FUNCTION_BLOCK Stage4 (* Template for a Basic Function Block Type *)
  (* Standard: 61499-2 *)
  (* Version 1.0, 2021-06-20, HP *)
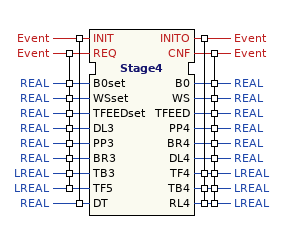
  EVENT_INPUT
    INIT WITH DT; (* Initialization Request *)
    REQ WITH B0set, WSset, TFEEDset, DL3, PP3, BR3, TB3, TF5; (* Normal Execution Request *)
  END_EVENT
  EVENT_OUTPUT
    INITO WITH TB4, TF4, RL4; (* Initialization Confirm *)
    CNF WITH TB4, DL4, TF4, BR4, PP4, RL4, B0, WS, TFEED; (* Execution Confirmation *)
  END_EVENT
  VAR_INPUT
    B0set : REAL;
    WSset : REAL;
    TFEEDset : REAL;
    DL3 : REAL;
    PP3 : REAL;
    BR3 : REAL;
    TB3 : LREAL;
    TF5 : LREAL;
    DT : REAL;
  END_VAR
  VAR_OUTPUT
    B0 : REAL;
    WS : REAL;
    TFEED : REAL;
    PP4 : REAL;
    BR4 : REAL;
    DL4 : REAL;
    TF4 : LREAL;
    TB4 : LREAL;
    RL4 : LREAL;
  END_VAR
  VAR
    AB : REAL; (* internal variabel *)
    UU : REAL;
    TREF : REAL;
    AD : REAL;
    AHC : REAL;
    AHR : REAL;
    AS : REAL;
    REC : REAL;
    WN : REAL;
    WN_1 : REAL;
    XKN : REAL;
    C1 : REAL;
    HS : REAL;
    G : REAL;
    W1 : REAL;
    TFREC : REAL;
    TS : REAL;
    DTS : REAL;
    TF4_last : REAL;
    RL4_last : REAL;
    TB4_last : REAL;
    USS : REAL;
    RHOB : REAL;
    CPB : REAL;
    CPF : REAL;
    FMW : REAL;
    HLV : REAL;
    HV : REAL;
    BPR : REAL;
    FMC : REAL;
    U : REAL;
    A : REAL;
    B : REAL;
    C : REAL;
    D1 : REAL;
    d : REAL;
    a : REAL;
    A1 : REAL;
    A2 : REAL;
    A3 : REAL;
    A4 : REAL;
    A5 : REAL;
    A6 : REAL;
    p : REAL;
    q : REAL;
    TC : REAL;
    PC : REAL;
    DTB4 : REAL;
    DEN4 : REAL;
    DH4 : REAL;
    DP4 : REAL;
    DPDH4 : REAL;
    DT4 : REAL;
    m : REAL;
    n : REAL;
    VR4 : REAL;
    DELTA4 : REAL;
    DELTA26 : REAL;
    DELTA48 : REAL;
    DELTA4_last : REAL;
    DELTA26_last : REAL;
    DELTA48_last : REAL;
  END_VAR
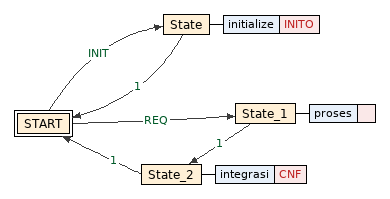
  EC_STATES
    START; (* Initial State *)
    State : initialize -> INITO;
    State_1 : proses;
    State_2 : integrasi -> CNF;
  END_STATES
  EC_TRANSITIONS
    START TO State := INIT;
    State TO START := 1;
    START TO State_1 := REQ;
    State_1 TO State_2 := 1;
    State_2 TO START := 1;
  END_TRANSITIONS
  ALGORITHM initialize IN ST: (* Initialization algorithm *)
TREF :=273.15;
AB :=57.2727;
AHC :=4069.2;
AHR :=2639.7;
AS :=3225.7;
REC :=0.0;
//TF2:=TF2;

//TFEED :=TFEED1+TREF;
 //TS:=TS1+TREF;
WN :=3.0;
XKN :=0.68;
HS:=0.11;
G :=9.81;
W1 :=0.50;

RL4 := 0.533784719363857;
TB4 := 356.263388068397;
TF4 := 352.376032234529;
TF5 := 349.772691418052;


RL4_last :=RL4;
TB4_last :=TB4;
TF4_last :=TF4;
  END_ALGORITHM
  ALGORITHM proses IN ST: (* kalkulasi *)
B0 :=B0set;
WS :=WSset;
TFEED:=TFEEDset;
UU := TFEEDset;
U :=UU;

USS :=49.767;
C1 :=0.625;
RHOB :=1032.4; //maassa jenis brine
CPB :=1.00; //heatcapacity Brine
CPF :=1.00; //heat capacity feed
FMW :=23654.0;
HLV :=563.7959;
HV :=625.1971;
BPR :=2.192;
FMC :=34736.09;
//U :=UU; //feed temp



///  Calculate the physical properties

//A :=3.2437814;
//B :=5.86826*0.001;
//C :=1.1702379*0.00000001;
//D1 :=2.1878462*0.001;
//TC :=647.27;
//PC :=218.167;


A1 :=3.2437814;
A2:=5.86826*0.001;
A3:=1.1702379*0.00000001;
A4 :=2.1878462*0.001;
A5 :=647.27;
A6 :=218.167;

DTB4 :=A5-TB4;
DEN4 :=(A1+A2*DTB4+A3*DTB4*DTB4*DTB4)/(1+A4*DTB4)*DTB4/TB4;
p:=DEN4;
q:=10.0;
PP4 :=A6/(EXPT(q, p));

// calculate the brine flow rates
DP4:=PP3-PP4;
DH4:=RL4-C1*HS;
DPDH4 :=DP4*101000+G*RHOB*DH4;
m:=DPDH4*RHOB;
n:=0.5;
BR4 :=WN*XKN*RL4*(EXPT(m, n));
BR4 :=BR4*60.0/1000.0;

// calculate the vapor flow rates

DT4 :=TB4-BPR/1.8-(TF5+TF4)*0.5;
VR4 :=U*AHC*DT4/HLV/1000.0;
DL4 :=DL3+VR4;


//// state equation
DELTA4 :=(BR3-BR4-VR4)*1000.0/RHOB/AB;
DELTA26 :=((BR3*CPB*(TB3-TB4))-VR4*(HV-CPB*(TB4-TREF)))*1000.0/AB/RHOB/CPB/RL4;
//DELTA23 :=DELTA23-VR1*(HV-CPB*(TB1-TREF));
//DELTA23 :=DELTA23*1000.0/AB/RHOB/CPB/RL1;

DELTA48 :=((B0*CPF*(TF5-TF4)*1000+(U*AHC*DT4)))/FMW/CPF;
//DELTA45 :=DELTA45+;
//DELTA45 :=DELTA45/FMW/CPF;
  END_ALGORITHM
  ALGORITHM integrasi IN ST: (* new algorithm *)
B0 :=B0set;
WS :=WSset;
TFEED:=TFEEDset;
//integrasi
RL4 := (DELTA4 + DELTA4_last)*0.5*DT + RL4_last;
DELTA4_last :=DELTA4 ;
RL4_last :=RL4;

TB4 := (DELTA26 + DELTA26_last)*0.5*DT + TB4_last;
DELTA26_last :=DELTA26 ;
TB4_last:=TB4;

TF4 := (DELTA48 + DELTA48_last)*0.5*DT + TF4_last;
DELTA48_last :=DELTA48 ;
TF4_last :=TF4;
  END_ALGORITHM
END_FUNCTION_BLOCK
